(* IEC 61131-3 sources: Industry-PLC-LLM/data/PLCBEAD_repo/PLCBEAD_PLCEmbed-main/PLC-BEAD/Source/GEB/WORD_OF_DWORD, 1 file *)

(* ---- WORD_OF_DWORD.ST ---- *)
FUNCTION _BYTE_TO_INT:INT
	VAR_INPUT
		IN :	BYTE;
	END_VAR

	_BYTE_TO_INT := USINT_TO_INT(BYTE_TO_USINT(IN));
END_FUNCTION

FUNCTION WORD_OF_DWORD:WORD
	VAR_INPUT
		IN: DWORD;
		N :	BYTE;
	END_VAR
	WORD_OF_DWORD := DWORD_TO_WORD(SHR(IN,_BYTE_TO_INT(SHL(n,4))));
END_FUNCTION

PROGRAM program0
  	VAR
		IN :	DWORD;
		N :	BYTE;
		CEIL5_OUT : WORD;
	  END_VAR

  	CEIL5_OUT := WORD_OF_DWORD(IN, N);
END_PROGRAM
